TYPE SubIndexModuleBase :
STRUCT
	SubIndex : STRING;
	SizeByte  : UDINT;
END_STRUCT
END_TYPE

(* stored: Version 1.1.0.1, ProductVersion 3.1.4024.3
   DUT SubIndexModuleBase: Id {54fee83e-ef9e-4aae-bdd1-b45935106ee0} *)
